// TIA Portal V21 export
DATA_BLOCK "BATCH LINE PRINT_DB"   // DB14
// stored: InstanceOfName BATCH LINE PRINT, InstanceOfType FB
"BATCH LINE PRINT"
   // VAR_INPUT
   //    PrintInetrval : Int;
   //    SecPulse : Bool;
   // END_VAR
   // VAR_IN_OUT
   //    ResetBatchTimer : Bool;
   //    BatchSelected : Bool;
   // END_VAR
   // VAR
   //    IEC_Counter_0_Instance { S7_SetPoint := 'True'} : CTU_INT;
   // END_VAR
BEGIN
END_DATA_BLOCK
